(* IEC 61131-3 sources: Conveyor/test/Conveyor, 12 files *)

(* ---- ConveyorAutoStartupTest.st ---- *)
USING Simatic.Ax.Conveyor.Mocks;
USING Simatic.Ax.Conveyor;
USING AxUnit.Assert;
USING Simatic.Ax.AutomationBase;
USING MotorTests.Mocks;

NAMESPACE Simatic.Ax.Conveyor
    /// Tests for conveyor automatic startup behavior
    /// Verifies startup sequences, release conditions, and motor control during startup
    {TestFixture}
    CLASS ConveyorAutoStartupTest
        VAR
            conv : ConveyorBase;
            convStateless : ConveyorBase;
            mockMan : MockOperatingMode := (Mode := OperatingModes#Manual);
            mockManStateless : MockOperatingMode := (Mode := OperatingModes#Manual);
            relTrue : MockIsReleased_TRUE;
            relTrueStateless : MockIsReleased_TRUE;
            relFalse : MockIsReleased_FALSE;
            relFalseStateless : MockIsReleased_FALSE;
            autoStart : MockAutoStartup;
            autoStartStateless : MockAutoStartup;
            sensorMockQ_QRis_True : MockBinSignal := (QValue := TRUE, QRisValue := TRUE, QFalValue := FALSE);
            sensorMockQ_True : MockBinSignal := (QValue := TRUE, QRisValue := FALSE, QFalValue := FALSE);
            sensorMockQ_False : MockBinSignal := (QValue := FALSE, QRisValue := FALSE, QFalValue := FALSE);
            mockMotor : MockMotor;
            mockMotorStateless : MockMotor;
        END_VAR

        {TestSetup}
        METHOD PUBLIC Setup
            // Initialize stateless instances for each test
            conv := convStateless;
            mockMan := mockManStateless;
            relTrue := relTrueStateless;
            relFalse := relFalseStateless;
            autoStart := autoStartStateless;
            mockMotor := mockMotorStateless;
            mockMotor.Reset();
        END_METHOD

        {Test}
        METHOD PUBLIC Conveyor_Is_Stopped_InAutomatic_Without_Release
            // Arrange - Setup conveyor in automatic mode without release
            mockMan.mode := OperatingModes#Automatic;
            conv.Mode := mockMan;
            conv.Motor := mockMotor;
            conv.ExternalRelease := relTrue;
            conv.ExternalAutoStartup := autoStart;
            conv.StopSensor := sensorMockQ_False;
            autoStart.startupStatus := StartUpStatus#NotReleased;  // Not released

            // Verify setup is valid
            Equal(expected := FALSE, actual := HasConfigErrorTest(conv));

            // Act - Run cyclic execution
            conv.RunCyclic();

            // Assert - Motor should not be running without release
            Equal(expected := FALSE, actual := mockMotor.IsRunning());
        END_METHOD
        {Test}
        METHOD PUBLIC Conveyor_Is_Stopped_WhileStartingUp
            // Arrange - Setup conveyor during startup phase
            mockMan.mode := OperatingModes#Automatic;
            conv.Mode := mockMan;
            conv.Motor := mockMotor;
            conv.ExternalRelease := relTrue;
            autoStart.startupStatus := StartUpStatus#AutoStartingUp;  // Still starting up
            conv.StopSensor := sensorMockQ_False;
            conv.ExternalAutoStartup := autoStart;

            // Verify setup is valid
            Equal(expected := FALSE, actual := HasConfigErrorTest(conv));

            // Act - Run cyclic execution
            conv.RunCyclic();

            // Assert - Motor should not run during startup phase
            Equal(expected := FALSE, actual := mockMotor.IsRunning());
        END_METHOD
        {Test}
        METHOD PUBLIC Conveyor_Starts_After_AutoRelease
            // Arrange - Setup conveyor with auto-release completed
            mockMan.mode := OperatingModes#Automatic;
            conv.Mode := mockMan;
            conv.Motor := mockMotor;
            conv.ExternalRelease := relTrue;
            conv.StopSensor := sensorMockQ_False;
            autoStart.startupStatus := StartUpStatus#AutoStartedUp;  // Fully started up
            conv.ExternalAutoStartup := autoStart;

            // Mock timer to pass through immediately
            AxUnit.Mocking.Mock(NAME_OF(System.Timer.OffDelay), NAME_OF(Simatic.Ax.Mocks.OffDelayMock_pass_trough));

            // Act - Run cyclic execution
            conv.RunCyclic();

            // Assert - Motor should be running after auto-release
            Equal(expected := TRUE, actual := mockMotor.IsRunning());
        END_METHOD
        {Test}
        METHOD PUBLIC Conveyor_Stopps_after_loosing_release
            // Arrange - First start conveyor, then lose release
            THIS.Conveyor_Starts_After_AutoRelease();
            autoStart.startupStatus := StartUpStatus#NotReleased;  // Lose release

            // Verify setup is valid
            Equal(expected := FALSE, actual := HasConfigErrorTest(conv));

            // Act - Run cyclic execution after losing release
            conv.RunCyclic();

            // Assert - Motor should stop after losing release
            Equal(expected := FALSE, actual := mockMotor.IsRunning());
        END_METHOD
    END_CLASS

END_NAMESPACE

(* ---- ConveyorManualModeTest.st ---- *)
USING Simatic.Ax.Conveyor.Mocks;
USING Simatic.Ax.Conveyor;
USING AxUnit.Assert;
USING Simatic.Ax.AutomationBase;
USING MotorTests.Mocks;

NAMESPACE Simatic.Ax.Conveyor

    /// Tests for conveyor manual mode operation
    /// Verifies manual start/stop behavior, release conditions, and mode transitions
    {TestFixture}
    CLASS TestConveyorManualMode
        VAR
            conv : ConveyorBase;
            convStateless : ConveyorBase;
            mockMan : MockOperatingMode;
            mockManStateless : MockOperatingMode;
            relTrue : MockIsReleased_TRUE;
            relTrueStateless : MockIsReleased_TRUE;
            relFalse : MockIsReleased_FALSE;
            relFalseStateless : MockIsReleased_FALSE;
            StopSensor : MockBinSignal := (QValue := TRUE);
            mockMotor : MockMotor;
            mockMotorStateless : MockMotor;
        END_VAR

        {TestSetup}
        METHOD PUBLIC Setup
            // Initialize stateless instances for each test
            conv := convStateless;
            mockMan := mockManStateless;
            relTrue := relTrueStateless;
            relFalse := relFalseStateless;
            mockMotor := mockMotorStateless;
            mockMotor.Reset();
        END_METHOD

        {Test}
        METHOD PUBLIC ConveyorIsStoppedByDefault
            // Arrange - Setup conveyor in automatic mode with release
            conv.StopSensor := StopSensor;
            conv.Motor := mockMotor;
            mockMan.mode := OperatingModes#Automatic;
            conv.Mode := mockMan;
            conv.ExternalRelease := relTrue;

            // Verify configuration is valid
            Equal(expected := FALSE, actual := HasConfigErrorTest(conv));

            // Act - Run cyclic execution twice
            conv.RunCyclic();

            // Assert - Motor should remain stopped without explicit start command
            Equal(expected := FALSE, actual := mockMotor.IsRunning());

            // Act - Run cyclic again
            conv.RunCyclic();

            // Assert - Motor should still be stopped
            Equal(expected := FALSE, actual := mockMotor.IsRunning());
        END_METHOD
        {Test}
        METHOD PUBLIC Conveyor_InManualMode_RunReleasedOnManualStart
            // Arrange - Setup conveyor in manual mode with release
            conv.StopSensor := StopSensor;
            conv.Motor := mockMotor;
            conv.Mode := mockMan;  // Default mode is Manual
            conv.ExternalRelease := relTrue;

            // Act - Issue manual start command and run cyclic
            conv.StartManual();
            conv.RunCyclic();

            // Assert - Motor should be running after manual start
            Equal(expected := TRUE, actual := mockMotor.IsRunning());
        END_METHOD
        {Test}
        METHOD PUBLIC NotReleased_Conveyor_DoNotSetRunRelease
            // Arrange - Setup conveyor without release signal
            conv.StopSensor := StopSensor;
            conv.Motor := mockMotor;
            conv.Mode := mockMan;
            conv.ExternalRelease := relFalse;  // No release signal

            // Verify configuration is valid
            Equal(expected := FALSE, actual := HasConfigErrorTest(conv));

            // Act - Run cyclic, then issue manual start, then run cyclic again
            conv.RunCyclic();
            conv.StartManual();
            conv.RunCyclic();

            // Assert - Motor should not run without release signal
            Equal(expected := FALSE, actual := mockMotor.IsRunning());
        END_METHOD
        {Test}
        METHOD PUBLIC ConveyorManualRunning_Stops_when_release_signal_has_left
            // Arrange - Setup conveyor running in manual mode
            conv.StopSensor := StopSensor;
            conv.Motor := mockMotor;
            THIS.Conveyor_InManualMode_RunReleasedOnManualStart();

            // Act - Run cyclic while motor is running
            conv.RunCyclic();

            // Assert - Motor should still be running
            Equal(expected := TRUE, actual := mockMotor.IsRunning());

            // Act - Run cyclic again
            conv.RunCyclic();

            // Assert - Motor should still be running
            Equal(expected := TRUE, actual := mockMotor.IsRunning());

            // Act - Remove release signal and run cyclic
            conv.ExternalRelease := relFalse;
            conv.RunCyclic();

            // Assert - Motor should stop when release signal is lost
            Equal(expected := FALSE, actual := mockMotor.IsRunning());
        END_METHOD
        {Test}
        METHOD PUBLIC Conveyor_InAutomaticMode_IsNotRunReleasedOnManualStart
            // Arrange - Setup conveyor in automatic mode with release
            conv.StopSensor := StopSensor;
            conv.Motor := mockMotor;
            mockMan.mode := OperatingModes#Automatic;
            conv.Mode := mockMan;
            conv.ExternalRelease := relTrue;

            // Verify configuration is valid
            Equal(expected := FALSE, actual := HasConfigErrorTest(conv));

            // Act - Issue manual start command (should be ignored in automatic mode)
            conv.StartManual();
            conv.RunCyclic();

            // Assert - Motor should not run because manual start is ignored in automatic mode
            Equal(expected := FALSE, actual := mockMotor.IsRunning());
        END_METHOD
        {Test}
        METHOD PUBLIC ConveyorRunningInManualMode_Stops_on_Stop_Command
            // Arrange - Setup conveyor running in manual mode
            conv.StopSensor := StopSensor;
            conv.Motor := mockMotor;
            THIS.Conveyor_InManualMode_RunReleasedOnManualStart();

            // Act - Issue stop command and run cyclic
            conv.Stop();
            conv.RunCyclic();

            // Assert - Motor should stop after stop command
            Equal(expected := FALSE, actual := mockMotor.IsRunning());
        END_METHOD
    END_CLASS

END_NAMESPACE

(* ---- ConveyorMotorIntegrationTest.st ---- *)
USING AxUnit.Assert;
USING Simatic.Ax.Conveyor;
USING MotorTests.Mocks;

NAMESPACE ConveyorTests
    /// Integration tests for Conveyor with Motor
    {TestFixture}
    CLASS ConveyorMotorIntegrationTest
        VAR PROTECTED
            conveyor : ConveyorBase;
            conveyorStateless : ConveyorBase;
            motor : MockMotor;
            motorStateless : MockMotor;
        END_VAR

        {TestSetup}
        METHOD PUBLIC TestSetup
            conveyor := conveyorStateless;
            motor := motorStateless;
            motor.Reset();
        END_METHOD

        {Test}
        METHOD PUBLIC Test_ConveyorWithoutMotor_NoError
            // Arrange - No motor assigned

            // Act
            conveyor.RunCyclic();  // Init is now called automatically by RunCyclic

            // Assert - No motor calls when motor is NULL
            Equal(expected := 0, actual := motor.StartMotorCallCount);
        END_METHOD

        {Test}
        METHOD PUBLIC Test_ConveyorWithMotor_MotorInjected
            // Arrange
            conveyor.Motor := motor;

            // Act
            conveyor.RunCyclic();  // Init is now called automatically by RunCyclic

            // Assert - Motor is properly injected
            Equal(expected := TRUE, actual := (conveyor.Motor <> NULL));
        END_METHOD

        {Test}
        METHOD PUBLIC Test_MotorConfiguration_IsAccessible
            // Arrange & Act
            conveyor.Motor := motor;
            conveyor.AutomaticSpeed := 75.0;
            conveyor.Acceleration := 10.0;

            // Assert - Configuration is properly set
            Equal(expected := 75.0, actual := conveyor.AutomaticSpeed);
            Equal(expected := 10.0, actual := conveyor.Acceleration);
        END_METHOD

        {Test}
        METHOD PUBLIC Test_MotorConfiguration_SlowSpeed
            // Arrange
            conveyor.Motor := motor;
            conveyor.AutomaticSpeed := 75.0;
            conveyor.ManualSpeed := 30.0;

            // Act & Assert - Configuration is accessible
            Equal(expected := 75.0, actual := conveyor.AutomaticSpeed);
            Equal(expected := 30.0, actual := conveyor.ManualSpeed);
        END_METHOD

        {Test}
        METHOD PUBLIC Test_ConveyorStop_CallsStopMethod
            // Arrange
            conveyor.Motor := motor;
            Motor.StartMotor();

            // Act
            conveyor.Stop();

            // Assert - Stop method was called successfully
            Equal(expected := TRUE, actual := TRUE);  // Stop executed without error
        END_METHOD

        {Test}
        METHOD PUBLIC Test_IsMotorRunning_ReturnsMotorState
            // Arrange
            conveyor.Motor := motor;

            // Act & Assert - Motor not running
            Equal(expected := FALSE, actual := conveyor.ConveyorIsRunning());

            // Start motor
            Motor.StartMotor();

            // Act & Assert - Motor running
            Equal(expected := TRUE, actual := conveyor.ConveyorIsRunning());
        END_METHOD

        {Test}
        METHOD PUBLIC Test_MotorConfiguration_UsesCustomValues
            // Arrange
            conveyor.Motor := motor;
            conveyor.AutomaticSpeed := 80.0;
            conveyor.ManualSpeed := 25.0;
            conveyor.Acceleration := 15.0;
            conveyor.Deceleration := 20.0;

            // Act & Assert
            Equal(expected := 80.0, actual := conveyor.AutomaticSpeed);
            Equal(expected := 25.0, actual := conveyor.ManualSpeed);
            Equal(expected := 15.0, actual := conveyor.Acceleration);
            Equal(expected := 20.0, actual := conveyor.Deceleration);
        END_METHOD

        {Test}
        METHOD PUBLIC Test_MotorStopWithDeceleration
            // Arrange
            conveyor.Motor := motor;
            conveyor.Deceleration := 20.0;
            motor.FixedDeceleration := 20.0;
            Motor.StartMotor();

            // Act
            Motor.StopMotor();

            // Assert - Motor uses configured deceleration and stops
            Equal(expected := 20.0, actual := motor.FixedDeceleration);
            Equal(expected := FALSE, actual := motor.IsRunning());
        END_METHOD

        {Test}
        METHOD PUBLIC Test_IsMotorRunning_WithoutMotor_ReturnsFalse
            // Arrange
            conveyor.Motor := NULL;

            // Act & Assert
            Equal(expected := FALSE, actual := conveyor.ConveyorIsRunning());
        END_METHOD
    END_CLASS

    /// Tests for motor control logic
    {TestFixture}
    CLASS ConveyorMotorControlTest
        VAR PROTECTED
            conveyor : ConveyorBase;
            conveyorStateless : ConveyorBase;
            motor : MockMotor;
            motorStateless : MockMotor;
        END_VAR

        {TestSetup}
        METHOD PUBLIC TestSetup
            conveyor := conveyorStateless;
            motor := motorStateless;
            motor.Reset();
            conveyor.Motor := motor;
        END_METHOD

        {Test}
        METHOD PUBLIC Test_MockMotor_CanStartAndStop
            // Arrange
            conveyor.AutomaticSpeed := 75.0;
            conveyor.Deceleration := 15.0;

            // Act - Start motor
            Motor.StartMotor();

            // Assert - Motor started
            Equal(expected := TRUE, actual := motor.IsRunning());
            Equal(expected := 1, actual := motor.StartMotorCallCount);

            // Act - Stop motor
            Motor.StopMotor();

            // Assert - Motor stopped
            Equal(expected := FALSE, actual := motor.IsRunning());
            Equal(expected := 1, actual := motor.StopMotorCallCount);
        END_METHOD

        {Test}
        METHOD PUBLIC Test_MockMotor_TracksCallCounts
            // Arrange
            motor.TargetSpeed := 80.0;
            motor.FixedAcceleration := 12.0;
            motor.FixedDeceleration := 18.0;

            // Act
            Motor.StartMotor();
            Motor.StopMotor();

            // Assert - Call counts are tracked and properties are set
            Equal(expected := 1, actual := motor.StartMotorCallCount);
            Equal(expected := 1, actual := motor.StopMotorCallCount);
            Equal(expected := 80.0, actual := motor.TargetSpeed);
            Equal(expected := 12.0, actual := motor.FixedAcceleration);
            Equal(expected := 18.0, actual := motor.FixedDeceleration);
        END_METHOD

        {Test}
        METHOD PUBLIC Test_MockMotor_ResetClearsState
            // Arrange
            Motor.StartMotor();

            // Act
            motor.Reset();

            // Assert - All state cleared
            Equal(expected := FALSE, actual := motor.IsRunning());
            Equal(expected := 0, actual := motor.StartMotorCallCount);
            Equal(expected := 0, actual := motor.StopMotorCallCount);
            Equal(expected := 0.0, actual := motor.GetCurrentSpeed());
        END_METHOD
    END_CLASS
END_NAMESPACE

(* ---- ConveyorOccupiedStatus.st ---- *)
USING Simatic.Ax.Conveyor.Mocks;
USING Simatic.Ax.Conveyor;
USING AxUnit.Assert;
USING Simatic.Ax.AutomationBase;
USING MotorTests.Mocks;

NAMESPACE Simatic.Ax.Conveyor

    /// Tests for conveyor occupied status detection
    /// Verifies occupied state based on sensor coverage, operating mode, and startup status
    {TestFixture}
    CLASS ConveyorOccupiedStatus
        VAR
            conv : ConveyorBase;
            convStateless : ConveyorBase;
            mockOperatingMode : MockOperatingMode;
            mockOperatingModeStateless : MockOperatingMode;
            relTrue : MockIsReleased_TRUE;
            relTrueStateless : MockIsReleased_TRUE;
            relFalse : MockIsReleased_FALSE;
            relFalseStateless : MockIsReleased_FALSE;
            autoStart : MockAutoStartup;
            autoStartStateless : MockAutoStartup;
            sensorMockQ_QRis_True : MockBinSignal := (QValue := TRUE, QRisValue := TRUE, QFalValue := FALSE);
            sensorMockQ_True : MockBinSignal := (QValue := TRUE, QRisValue := FALSE, QFalValue := FALSE);
            sensorMockQ_False : MockBinSignal := (QValue := FALSE, QRisValue := FALSE, QFalValue := FALSE);
            convNext : MockingConveyor;
            convNextStateless : MockingConveyor;
            mockMotor : MockMotor;
            mockMotorStateless : MockMotor;
        END_VAR

        {TestSetup}
        METHOD PUBLIC Setup
            // Initialize stateless instances for each test
            conv := convStateless;
            mockOperatingMode := mockOperatingModeStateless;
            relTrue := relTrueStateless;
            relFalse := relFalseStateless;
            autoStart := autoStartStateless;
            convNext := convNextStateless;
            mockMotor := mockMotorStateless;
            mockMotor.Reset();
        END_METHOD

        METHOD PUBLIC SetupAutoStarted
            conv.StopSensor := sensorMockQ_False;
            conv.Motor := mockMotor;
            mockOperatingMode.mode := OperatingModes#Automatic;
            conv.Mode := mockOperatingMode;
            conv.Motor := mockMotor;
            conv.ExternalRelease := relTrue;
            conv.ExternalAutoStartup := autoStart;
            conv.NextConveyor := convNext;
            autoStart.startupStatus := StartUpStatus#AutoStartedUp;
        END_METHOD
        {Test}
        METHOD PUBLIC Conveyor_is_not_occupied_by_default
            // Arrange - Setup conveyor in auto-started state with no sensor coverage
            THIS.SetupAutoStarted();

            // Verify configuration is valid
            Equal(expected := FALSE, actual := HasConfigErrorTest(conv));

            // Act - Run cyclic execution
            conv.RunCyclic();

            // Assert - Conveyor should not be occupied without sensor coverage
            Equal(expected := FALSE, actual := conv.IsOccupied());
        END_METHOD
        {Test}
        METHOD PUBLIC Conveyor_Is_occupied_when_sensor_covered_and_automatic_is_on_while_next_is_not_rtr
            // Arrange - Setup conveyor in automatic mode with sensor covered
            THIS.SetupAutoStarted();
            conv.StopSensor := sensorMockQ_True;  // Sensor covered
            conv.Motor := mockMotor;
            // Next conveyor not ready to receive (default state)

            // Verify configuration is valid
            Equal(expected := FALSE, actual := HasConfigErrorTest(conv));

            // Act - Run cyclic execution
            conv.RunCyclic();

            // Assert - Conveyor should be occupied when sensor is covered in automatic mode
            Equal(expected := TRUE, actual := conv.IsOccupied());
        END_METHOD
        {Test}
        METHOD PUBLIC Conveyor_Ignores_occupied_state_when_in_manual
            // Arrange - Setup conveyor in manual mode with sensor covered
            THIS.SetupAutoStarted();
            conv.ExternalAutoStartup := NULL;
            conv.StopSensor := sensorMockQ_True;  // Sensor covered
            conv.Motor := mockMotor;
            mockOperatingMode.mode := OperatingModes#Manual;  // Manual mode

            // Verify configuration is valid
            Equal(expected := FALSE, actual := HasConfigErrorTest(conv));

            // Act - Run cyclic execution
            conv.RunCyclic();

            // Assert - Conveyor should not report occupied in manual mode (occupied detection disabled)
            Equal(expected := FALSE, actual := conv.IsOccupied());

        END_METHOD

        {Test}
        METHOD PUBLIC Conveyor_Is_occupied_when_sensor_covered_and_switch_to_automatic_while_next_is_not_rtr
            // Arrange - Setup conveyor with sensor covered, starting in manual mode
            conv.StopSensor := sensorMockQ_True;  // Sensor covered
            conv.Motor := mockMotor;
            mockOperatingMode.mode := OperatingModes#Manual;
            conv.Mode := mockOperatingMode;
            conv.ExternalRelease := relTrue;
            conv.ExternalAutoStartup := autoStart;
            conv.NextConveyor := convNext;

            // Act - Test in NotReleased state (manual mode)
            autoStart.startupStatus := StartUpStatus#NotReleased;
            conv.RunCyclic();

            // Assert - Not occupied in manual/not released state
            Equal(expected := FALSE, actual := conv.IsOccupied());

            // Act - Test during startup sequence
            autoStart.startupStatus := StartUpStatus#AutoStartingUp;
            conv.RunCyclic();

            // Assert - Not occupied during startup
            Equal(expected := FALSE, actual := conv.IsOccupied());

            // Act - Complete startup to automatic mode
            autoStart.startupStatus := StartUpStatus#AutoStartedUp;
            conv.RunCyclic();

            // Assert - Now occupied after fully started in automatic mode
            Equal(expected := TRUE, actual := conv.IsOccupied());
        END_METHOD
    END_CLASS

END_NAMESPACE

(* ---- ConveyorResetTest.st ---- *)
USING Simatic.Ax.AutomationBase;
USING AxUnit.Assert;
USING Simatic.Ax.Conveyor;
USING Simatic.Ax.Conveyor.Mocks;
USING Simatic.Ax.AutomationBase;
USING MotorTests.Mocks;

NAMESPACE Simatic.Ax.Conveyor.Tests

    {TestFixture}
    CLASS ConveyorResetTest
        VAR
            conveyor : ConveyorBase;
            conveyorStateless : ConveyorBase;
            mockMotor : MockMotor;
            mockMotorStateless : MockMotor;
            mockMode : MockOperatingMode := (Mode := OperatingModes#Manual);
            mockModeStateless : MockOperatingMode := (Mode := OperatingModes#Manual);
            mockRelease : MockIsReleased_TRUE;
            mockReleaseStateless : MockIsReleased_TRUE;
            mockAutoStartup : MockAutoStartup;
            mockAutoStartupStateless : MockAutoStartup;
            mockResetManager : MockResetManager;
            mockResetManagerStateless : MockResetManager;
            sensorMockQ_True : MockBinSignal := (QValue := TRUE, QRisValue := FALSE, QFalValue := FALSE);
            sensorMockQ_False : MockBinSignal := (QValue := FALSE, QRisValue := FALSE, QFalValue := FALSE);
        END_VAR

        {TestSetup}
        METHOD PUBLIC Setup
            // Reset to stateless instances for test isolation
            conveyor := conveyorStateless;
            mockMotor := mockMotorStateless;
            mockMotor.Reset();
            mockMode := mockModeStateless;
            mockRelease := mockReleaseStateless;
            mockAutoStartup := mockAutoStartupStateless;
            mockResetManager := mockResetManagerStateless;
            mockResetManager.Reset();

            // Configure conveyor
            conveyor.StopSensor := sensorMockQ_False;
            conveyor.Motor := mockMotor;
            conveyor.ExternalRelease := mockRelease;
            conveyor.Mode := mockMode;
            conveyor.ExternalAutoStartup := mockAutoStartup;
            conveyor.ResetCommand := mockResetManager;

            // Set default states
            mockMode.mode := OperatingModes#Automatic;
            mockAutoStartup.startupStatus := StartUpStatus#AutoStartedUp;

            // Initialize conveyor by calling RunCyclic (triggers InitUser)
            conveyor.RunCyclic();
        END_METHOD

        {Test}
        METHOD PUBLIC Test_ResetFault_ClearsManualStartFlag
            // Arrange
            mockMode.mode := OperatingModes#Manual;
            mockAutoStartup.startupStatus := StartUpStatus#Manual;
            conveyor.RunCyclic();
            conveyor.StartManual();
            conveyor.RunCyclic();
            Equal(expected := TRUE, actual := Conveyor.ConveyorIsRunning());
            conveyor.SetError(errorState := WORD#16#8199, errorText := 'any error');

            // Verify motor is running
            Equal(expected := TRUE, actual := mockMotor.StartMotorCallCount > 0);

            // Act - trigger reset via ResetManager
            mockResetManager.ResetCommandActive := TRUE;
            conveyor.RunCyclic();

            // Assert - manual start flag should be cleared
            mockResetManager.ResetCommandActive := FALSE;
            conveyor.RunCyclic();
            Equal(expected := TRUE, actual := mockMotor.StopMotorCallCount > 0);
        END_METHOD

        {Test}
        METHOD PUBLIC Test_ResetFault_AllowsAutoRestart
            // Arrange - setup conveyor with material
            conveyor.StopSensor := sensorMockQ_True;
            conveyor.RunCyclic();

            // Simulate error
            conveyor.SetError(errorState := WORD#16#8001, errorText := 'Test error');

            // Act - trigger reset via ResetManager
            mockResetManager.ResetCommandActive := TRUE;
            conveyor.RunCyclic();

            // Assert - conveyor should be able to auto-restart after reset
            // The auto-release flags are NOT cleared, allowing automatic restart
            mockResetManager.ResetCommandActive := FALSE;
            conveyor.RunCyclic();
            conveyor.TriggerStartInAutomatic();
            conveyor.RunCyclic();
            Equal(expected := TRUE, actual := mockMotor.StartMotorCallCount > 0);
        END_METHOD

        {Test}
        METHOD PUBLIC Test_ResetFault_AllowsNormalOperationAfterReset
            // Arrange - trigger reset
            mockResetManager.ResetCommandActive := TRUE;
            conveyor.RunCyclic();
            mockResetManager.ResetCommandActive := FALSE;

            // Act - simulate normal operation
            conveyor.StopSensor := sensorMockQ_True;
            conveyor.RunCyclic();
            conveyor.TriggerStartInAutomatic();
            conveyor.RunCyclic();

            // Assert - conveyor should be able to start normally
            Equal(expected := TRUE, actual := mockMotor.StartMotorCallCount > 0);
        END_METHOD

        {Test}
        METHOD PUBLIC Test_ResetFault_CanBeCalledMultipleTimes
            // Act - trigger reset multiple times via ResetManager
            mockResetManager.ResetCommandActive := TRUE;
            conveyor.RunCyclic();
            conveyor.RunCyclic();
            conveyor.RunCyclic();

            // Assert - should not cause any issues
            mockResetManager.ResetCommandActive := FALSE;
            conveyor.RunCyclic();
            Equal(expected := FALSE, actual := conveyor.HasError());
        END_METHOD
        {Test}
        METHOD PUBLIC Test_ResetFault_WithNullMotor_DoesNotCrash
            // Arrange
            conveyor.Motor := NULL;

            // Act & Assert - should not crash when reset is triggered
            mockResetManager.ResetCommandActive := TRUE;
            conveyor.RunCyclic();
            mockResetManager.ResetCommandActive := FALSE;
            conveyor.RunCyclic();
            Equal(expected := FALSE, actual := conveyor.HasError());
        END_METHOD

        {Test}
        METHOD PUBLIC Test_ResetFault_ClearsErrorState
            // Arrange - simulate an error condition
            conveyor.SetError(errorState := WORD#16#8001, errorText := 'Test error');
            Equal(expected := TRUE, actual := conveyor.HasError());

            // Act - trigger reset via ResetManager
            mockResetManager.ResetCommandActive := TRUE;
            conveyor.RunCyclic();

            // Assert - error should be cleared
            Equal(expected := FALSE, actual := conveyor.HasError());
        END_METHOD

        // {Test}
        // METHOD PUBLIC Test_ResetFault_BlockedWhenSensorStillCovered
        //     // Arrange - simulate sensor blocked during delivering
        //     sensorMockQ_True.QValue := TRUE;
        //     conveyor.StopSensor := sensorMockQ_True;
        //     conveyor.RunCyclic();
        //     conveyor.TriggerStartInAutomatic();
        //     conveyor.RunCyclic();

        //     // Simulate error condition
        //     conveyor.SetError(errorState := WORD#16#8001, errorText := 'Sensor blocked');
        //     Equal(expected := TRUE, actual := conveyor.HasError());

        //     // Act - try to reset while sensor is still covered via ResetManager
        //     mockResetManager.ResetCommandActive := TRUE;
        //     conveyor.RunCyclic();

        //     // Assert - error should NOT be cleared because sensor is still blocked
        //     Equal(expected := TRUE, actual := conveyor.HasError());
        // END_METHOD

        {Test}
        METHOD PUBLIC Test_ResetFault_AllowedWhenSensorCleared
            // Arrange - simulate sensor blocked, then cleared
            sensorMockQ_True.QValue := TRUE;
            conveyor.StopSensor := sensorMockQ_True;
            conveyor.RunCyclic();
            conveyor.TriggerStartInAutomatic();
            conveyor.RunCyclic();

            // Simulate error condition
            conveyor.SetError(errorState := WORD#16#8001, errorText := 'Sensor blocked');
            Equal(expected := TRUE, actual := conveyor.HasError());

            // Clear the sensor
            conveyor.StopSensor := sensorMockQ_False;
            conveyor.RunCyclic();

            // Act - reset after sensor is cleared via ResetManager
            mockResetManager.ResetCommandActive := TRUE;
            conveyor.RunCyclic();

            // Assert - error should be cleared now
            Equal(expected := FALSE, actual := conveyor.HasError());
        END_METHOD
    END_CLASS

END_NAMESPACE

(* ---- EndOfLineConveyorTest.st ---- *)
USING Simatic.Ax.Conveyor.Mocks;
USING Simatic.Ax.Conveyor;
USING AxUnit.Assert;
USING Simatic.Ax.AutomationBase;
USING MotorTests.Mocks;

NAMESPACE Simatic.Ax.Conveyor

    /// Tests for end-of-line conveyor behavior with NullReceiver
    /// Verifies that the last conveyor in a line can complete transfers without a next conveyor
    {TestFixture}
    CLASS EndOfLineConveyorTest
        VAR
            conv : ConveyorBase;
            convStateless : ConveyorBase;
            sensor : MockBinSignal;
            sensorStateless : MockBinSignal;
            relTrue : MockIsReleased_TRUE;
            relTrueStateless : MockIsReleased_TRUE;
            autoStart : MockAutoStartup := (startupStatus := StartUpStatus#AutoStartedUp);
            autoStartStateless : MockAutoStartup := (startupStatus := StartUpStatus#AutoStartedUp);
            mode : MockOperatingMode;
            modeStateless : MockOperatingMode;
            mockMotor : MockMotor;
            mockMotorStateless : MockMotor;
            nullReceiver : NullReceiver;
            nullReceiverStateless : NullReceiver;
        END_VAR

        {TestSetup}
        METHOD PUBLIC TestSetup
            // Initialize stateless instances for each test
            conv := convStateless;
            sensor := sensorStateless;
            relTrue := relTrueStateless;
            autoStart := autoStartStateless;
            mode := modeStateless;
            mockMotor := mockMotorStateless;
            mockMotor.Reset();
            nullReceiver := nullReceiverStateless;

            // Setup end-of-line conveyor (no NextConveyor configured)
            conv.NextConveyor := NULL;  // End of line - will use NullReceiver
            conv.StopSensor := sensor;
            conv.Motor := mockMotor;
            conv.ExternalRelease := relTrue;
            conv.ExternalAutoStartup := autoStart;
            conv.Mode := mode;
            mode.mode := OperatingModes#Automatic;
            conv.OffDelayTime := T#2s;
            AxUnit.Mocking.Mock('System.Timer.OffDelay', 'Simatic.Ax.Mocks.OffDelayMock_pass_trough');
        END_METHOD

        {Test}
        METHOD PUBLIC EndOfLine_conveyor_starts_transfer_when_sensor_covered
            // Arrange - End of line conveyor with no next conveyor
            sensor.QValue := FALSE;

            // Act - Run cyclic to initialize
            conv.RunCyclic();

            // Act - Item arrives on sensor
            sensor.QValue := TRUE;
            conv.RunCyclic();

            // Assert - Conveyor should start transfer even without next conveyor
            Equal(expected := TRUE, actual := conv.IsOccupied());
            Equal(expected := TRUE, actual := conv.DeliverStatus() = DeliverState#Delivering);
            Equal(expected := TRUE, actual := mockMotor.IsRunning());
        END_METHOD

        {Test}
        METHOD PUBLIC EndOfLine_conveyor_continues_running_until_item_leaves
            // Arrange - Start with item on sensor
            THIS.EndOfLine_conveyor_starts_transfer_when_sensor_covered();

            // Assert - Motor should be running
            Equal(expected := TRUE, actual := mockMotor.IsRunning());

            // Act - Continue running while item is on sensor
            conv.RunCyclic();
            Equal(expected := TRUE, actual := mockMotor.IsRunning());

            conv.RunCyclic();
            Equal(expected := TRUE, actual := mockMotor.IsRunning());

            // Act - Item leaves sensor (transfer complete)
            sensor.QValue := FALSE;
            conv.RunCyclic();

            // Assert - Transfer should be complete, motor still running due to off-delay
            Equal(expected := TRUE, actual := conv.DeliverStatus() = DeliverState#Idle);
            Equal(expected := FALSE, actual := conv.IsOccupied());
            Equal(expected := TRUE, actual := mockMotor.IsRunning());
        END_METHOD

        {Test}
        METHOD PUBLIC EndOfLine_conveyor_stops_after_offdelay_expires
            // Arrange - Complete transfer and wait for off-delay
            THIS.EndOfLine_conveyor_continues_running_until_item_leaves();

            // Assert - Motor still running after transfer
            Equal(expected := TRUE, actual := mockMotor.IsRunning());

            // Act - Simulate off-delay timer expiring
            AxUnit.Mocking.Mock('System.Timer.OffDelay', 'Simatic.Ax.Mocks.OffDelayMock_false');
            conv.RunCyclic();

            // Assert - Motor should stop after off-delay expires
            Equal(expected := FALSE, actual := mockMotor.IsRunning());
        END_METHOD
{Test}
METHOD PUBLIC NullReceiver_always_signals_ReadyToReceive
    // Arrange - NullReceiver already initialized in TestSetup

            // Act & Assert - NullReceiver should always return ReadyToReceive
            Equal(expected := TRUE, actual := nullReceiver.ReceiveStatus() = ReceiveState#ReadyToReceive);

            // Call multiple times to ensure consistent behavior
            Equal(expected := TRUE, actual := nullReceiver.ReceiveStatus() = ReceiveState#ReadyToReceive);
            Equal(expected := TRUE, actual := nullReceiver.ReceiveStatus() = ReceiveState#ReadyToReceive);
        END_METHOD
    END_CLASS

END_NAMESPACE

(* ---- ExtendRunningForConveyorTest.st ---- *)
USING Simatic.Ax.Conveyor.Mocks;
USING Simatic.Ax.Conveyor;
USING AxUnit.Assert;
USING Simatic.Ax.AutomationBase;
USING MotorTests.Mocks;

NAMESPACE Simatic.Ax.Conveyor

    /// Tests for extended running behavior of conveyor
    /// Verifies motor continues running after base position until timeout
    {TestFixture}
    CLASS ExtendRunningForConveyorTest
        VAR
            conv : ConveyorBase;
            convStateless : ConveyorBase;
            nextConv : MockingConveyor;
            nextConvStateless : MockingConveyor;
            sensor : MockBinSignal;
            sensorStateless : MockBinSignal;
            relTrue : MockIsReleased_TRUE;
            relTrueStateless : MockIsReleased_TRUE;
            relFalse : MockIsReleased_FALSE;
            relFalseStateless : MockIsReleased_FALSE;
            autoStart : MockAutoStartup := (startupStatus := StartUpStatus#AutoStartedUp);
            autoStartStateless : MockAutoStartup := (startupStatus := StartUpStatus#AutoStartedUp);
            mode : MockOperatingMode;
            modeStateless : MockOperatingMode;
            mockMotor : MockMotor;
            mockMotorStateless : MockMotor;
        END_VAR

        {TestSetup}
        METHOD PUBLIC TestSetup
            // Initialize stateless instances for each test
            conv := convStateless;
            nextConv := nextConvStateless;
            sensor := sensorStateless;
            relTrue := relTrueStateless;
            relFalse := relFalseStateless;
            autoStart := autoStartStateless;
            mode := modeStateless;
            mockMotor := mockMotorStateless;
            mockMotor.Reset();

            // Setup conveyor configuration
            conv.NextConveyor := nextConv;
            conv.StopSensor := sensor;
            conv.Motor := mockMotor;
            conv.ExternalRelease := relTrue;
            conv.Mode := mode;
        END_METHOD
        {Test}
        METHOD PUBLIC Conveyor_Stopps_after_base_position_run_after_timeout
            // Arrange - Setup conveyor in manual mode, not released
            conv.ExternalAutoStartup := autoStart;
            autoStart.startupStatus := StartUpStatus#NotReleased;

            // Mock timer to pass through immediately (no delay)
            AxUnit.Mocking.Mock('System.Timer.OffDelay', 'Simatic.Ax.Mocks.OffDelayMock_pass_trough');

            mode.mode := OperatingModes#Manual;
            sensor.QValue := FALSE;  // No item on sensor

            // Act - Run cyclic in manual mode
            conv.RunCyclic();

            // Assert - Motor should not be running in manual mode without release
            Equal(expected := FALSE, actual := mockMotor.IsRunning());

            // Act - Switch to automatic mode and complete startup
            mode.mode := OperatingModes#Automatic;
            autoStart.startupStatus := StartUpStatus#AutoStartedUp;
            conv.RunCyclic();

            // Assert - Motor should start running after switching to automatic with completed startup
            Equal(expected := TRUE, actual := mockMotor.IsRunning());
        END_METHOD
    END_CLASS

END_NAMESPACE

(* ---- MotorRunsDuringDeliveringTest.st ---- *)
USING Simatic.Ax.Conveyor.Mocks;
USING Simatic.Ax.Conveyor;
USING AxUnit.Assert;
USING Simatic.Ax.AutomationBase;
USING MotorTests.Mocks;

NAMESPACE Simatic.Ax.Conveyor

    /// Tests for motor behavior during Delivering state
    /// Verifies that motor continues running during transfer regardless of next conveyor state changes
    {TestFixture}
    CLASS MotorRunsDuringDeliveringTest
        VAR
            conv : ConveyorBase;
            convStateless : ConveyorBase;
            nextConv : MockingConveyor;
            nextConvStateless : MockingConveyor;
            sensor : MockBinSignal;
            sensorStateless : MockBinSignal;
            relTrue : MockIsReleased_TRUE;
            relTrueStateless : MockIsReleased_TRUE;
            autoStart : MockAutoStartup := (startupStatus := StartUpStatus#AutoStartedUp);
            autoStartStateless : MockAutoStartup := (startupStatus := StartUpStatus#AutoStartedUp);
            mode : MockOperatingMode;
            modeStateless : MockOperatingMode;
            mockMotor : MockMotor;
            mockMotorStateless : MockMotor;
        END_VAR

        {TestSetup}
        METHOD PUBLIC TestSetup
            // Initialize stateless instances for each test
            conv := convStateless;
            nextConv := nextConvStateless;
            sensor := sensorStateless;
            relTrue := relTrueStateless;
            autoStart := autoStartStateless;
            mode := modeStateless;
            mockMotor := mockMotorStateless;
            mockMotor.Reset();

            // Setup conveyor configuration
            conv.NextConveyor := nextConv;
            conv.StopSensor := sensor;
            conv.Motor := mockMotor;
            conv.ExternalRelease := relTrue;
            conv.ExternalAutoStartup := autoStart;
            conv.Mode := mode;
            mode.mode := OperatingModes#Automatic;
            conv.OffDelayTime := T#2s;
            AxUnit.Mocking.Mock('System.Timer.OffDelay', 'Simatic.Ax.Mocks.OffDelayMock_pass_trough');
        END_METHOD

        {Test}
        METHOD PUBLIC Motor_continues_running_during_Delivering_when_next_conveyor_changes_state
            // Arrange - Setup conveyor with sensor covered and next conveyor ready
            nextConv.RTR := ReceiveState#ReadyToReceive;
            sensor.QValue := TRUE;  // Item on sensor

            // Act - Run cyclic execution to start transfer
            conv.RunCyclic();

            // Assert - Motor should be running and transfer in progress
            Equal(expected := TRUE, actual := mockMotor.IsRunning());
            Equal(expected := TRUE, actual := conv.DeliverStatus() = DeliverState#Delivering);

            // Act - Next conveyor changes state to Receiving (simulating material arriving)
            nextConv.RTR := ReceiveState#Receiving;
            conv.RunCyclic();

            // Assert - Motor should STILL be running despite next conveyor state change
            Equal(expected := TRUE, actual := mockMotor.IsRunning());
            Equal(expected := TRUE, actual := conv.DeliverStatus() = DeliverState#Delivering);

            // Act - Continue running while sensor still covered (transfer ongoing)
            conv.RunCyclic();

            // Assert - Motor should continue running during transfer
            Equal(expected := TRUE, actual := mockMotor.IsRunning());
            Equal(expected := TRUE, actual := conv.DeliverStatus() = DeliverState#Delivering);
        END_METHOD

        {Test}
        METHOD PUBLIC Motor_continues_running_during_Delivering_over_multiple_cycles
            // Arrange - Setup conveyor with sensor covered and next conveyor ready
            nextConv.RTR := ReceiveState#ReadyToReceive;
            sensor.QValue := TRUE;  // Item on sensor

            // Act - Run cyclic execution to start transfer
            conv.RunCyclic();

            // Assert - Transfer should be in progress
            Equal(expected := TRUE, actual := conv.DeliverStatus() = DeliverState#Delivering);
            Equal(expected := TRUE, actual := mockMotor.IsRunning());

            // Act - Run multiple cycles while in Delivering
            conv.RunCyclic();
            Equal(expected := TRUE, actual := mockMotor.IsRunning());

            conv.RunCyclic();
            Equal(expected := TRUE, actual := mockMotor.IsRunning());

            conv.RunCyclic();
            Equal(expected := TRUE, actual := mockMotor.IsRunning());

            conv.RunCyclic();
            Equal(expected := TRUE, actual := mockMotor.IsRunning());

            // Assert - Motor should remain running throughout the transfer
            Equal(expected := TRUE, actual := conv.DeliverStatus() = DeliverState#Delivering);
        END_METHOD

        {Test}
        METHOD PUBLIC Motor_stops_only_after_transfer_completes_and_offdelay_expires
            // Arrange - Setup conveyor with sensor covered and next conveyor ready
            nextConv.RTR := ReceiveState#ReadyToReceive;
            sensor.QValue := TRUE;  // Item on sensor

            // Act - Run cyclic execution to start transfer
            conv.RunCyclic();
            Equal(expected := TRUE, actual := mockMotor.IsRunning());

            // Act - Item leaves sensor (transfer completes)
            sensor.QValue := FALSE;
            conv.RunCyclic();

            // Assert - Transfer should be complete, motor still running due to off-delay
            Equal(expected := TRUE, actual := conv.DeliverStatus() = DeliverState#Idle);
            Equal(expected := TRUE, actual := mockMotor.IsRunning());

            // Act - Simulate off-delay timer expiring
            AxUnit.Mocking.Mock('System.Timer.OffDelay', 'Simatic.Ax.Mocks.OffDelayMock_false');
            nextConv.RTR := ReceiveState#Idle;
            conv.RunCyclic();

            // Assert - Now motor should stop after off-delay expires
            Equal(expected := FALSE, actual := mockMotor.IsRunning());
        END_METHOD
    END_CLASS

END_NAMESPACE

(* ---- ReceiveFromPreviousConveyor.st ---- *)
USING Simatic.Ax.Conveyor.Mocks;
USING Simatic.Ax.Conveyor;
USING AxUnit.Assert;
USING Simatic.Ax.AutomationBase;
USING MotorTests.Mocks;

NAMESPACE Simatic.Ax.Conveyor

    /// Tests for receiving items from previous conveyor
    /// Verifies conveyor starts when previous conveyor signals ready to deliver or transfer in progress
    {TestFixture}
    CLASS ReceiveFromPreviousConveyor
        VAR
            conv, convStateless : ConveyorBase;
            nextConv, nextConvStateless : MockingConveyor;
            prevConv, prevConvStateless : MockingConveyor;
            sensor, sensorStateless : MockBinSignal;
            relTrue,  relTrueStateless : MockIsReleased_TRUE;
            relFalse, relFalseStateless : MockIsReleased_FALSE;
            autoStart, autoStartStateless : MockAutoStartup := (startupStatus := StartUpStatus#AutoStartedUp);
            mode, modeStateless : MockOperatingMode;
            mockMotor, mockMotorStateless : MockMotor;
        END_VAR

        {TestSetup}
        METHOD PUBLIC TestSetup
            // Initialize stateless instances for each test
            conv := convStateless;
            nextConv := nextConvStateless;
            prevConv := prevConvStateless;
            sensor := sensorStateless;
            relTrue := relTrueStateless;
            relFalse := relFalseStateless;
            autoStart := autoStartStateless;
            mode := modeStateless;
            mockMotor := mockMotorStateless;
            mockMotor.Reset();

            conv.NextConveyor := nextConv;
            conv.PrevConveyor := prevConv;
            conv.StopSensor := sensor;
            conv.Motor := mockMotor;
            conv.ExternalRelease := relTrue;
            conv.ExternalAutoStartup := autoStart;
            conv.StopSensor := sensor;
            conv.Motor := mockMotor;
            conv.Mode := mode;
            conv.Motor := mockMotor;
            mode.mode := OperatingModes#Automatic;
            AxUnit.Mocking.Mock('System.Timer.OffDelay', 'Simatic.Ax.Mocks.OffDelayMock_pass_trough');

        END_METHOD

        {Test}
        METHOD PUBLIC Idle_Conveyor_Starts_direct_On_Previous_Conveyor_is_ReadyToDeilver
            VAR_TEMP
                motorIsReleased : BOOL;
            END_VAR

            // Arrange - Setup conveyor with no sensor coverage, fully started
            sensor.QValue := FALSE;
            autoStart.startupStatus := StartUpStatus#AutoStartedUp;

            // Act - Run cyclic for initial home position run
            conv.RunCyclic();

            // Assert - Motor should be running for home position
            Equal(expected := TRUE, actual := mockMotor.IsRunning());

            // Act - Simulate home position run finished (off delay expires)
            AxUnit.Mocking.Mock('System.Timer.OffDelay', 'Simatic.Ax.Mocks.OffDelayMock_false');
            conv.RunCyclic();
            motorIsReleased := mockMotor.IsRunning();

            // Assert - Motor should stop after home position run completes
            Equal(expected := FALSE, actual := motorIsReleased);

            // Act - Previous conveyor announces ready to deliver
            AxUnit.Mocking.Mock('System.Timer.OffDelay', 'Simatic.Ax.Mocks.OffDelayMock_pass_trough');
            prevConv.RTD := DeliverState#ReadyToDeliver;
            conv.RunCyclic();

            // Assert - Motor should start immediately when previous conveyor is ready to deliver
            Equal(expected := TRUE, actual := mockMotor.IsRunning());

        END_METHOD

        {Test}
        METHOD PUBLIC Idle_Conveyor_Starts_direct_On_Previous_Conveyor_is_Delivering
            VAR_TEMP
                motorIsReleased : BOOL;
            END_VAR

            // Arrange - Setup conveyor with no sensor coverage, fully started
            sensor.QValue := FALSE;
            autoStart.startupStatus := StartUpStatus#AutoStartedUp;

            // Act - Run cyclic for initial home position run
            conv.RunCyclic();

            // Assert - Motor should be running for home position
            Equal(expected := TRUE, actual := mockMotor.IsRunning());

            // Act - Simulate home position run finished (off delay expires)
            AxUnit.Mocking.Mock('System.Timer.OffDelay', 'Simatic.Ax.Mocks.OffDelayMock_false');
            conv.RunCyclic();
            motorIsReleased := mockMotor.IsRunning();

            // Assert - Motor should stop after home position run completes
            Equal(expected := FALSE, actual := motorIsReleased);

            // Act - Previous conveyor announces transfer in progress
            AxUnit.Mocking.Mock('System.Timer.OffDelay', 'Simatic.Ax.Mocks.OffDelayMock_pass_trough');
            prevConv.RTD := DeliverState#Delivering;
            conv.RunCyclic();

            // Assert - Motor should start immediately when previous conveyor has transfer in progress
            Equal(expected := TRUE, actual := mockMotor.IsRunning());

        END_METHOD
    END_CLASS

END_NAMESPACE

(* ---- StopPositionTest.st ---- *)
USING Simatic.Ax.Conveyor.Mocks;
USING Simatic.Ax.Conveyor;
USING AxUnit.Assert;
USING Simatic.Ax.AutomationBase;

NAMESPACE Simatic.Ax.Conveyor

    /// Tests for stop position occupied detection
    /// Verifies occupied state based on sensor and equipment startup status
    {TestFixture}
    CLASS StopPositionTest
        VAR
            stop : StopPosition;
            stopStateless : StopPosition;
            sens : MockBinSignal;
            sensStateless : MockBinSignal;
            conv : MockingConveyor;
            convStateless : MockingConveyor;
            eq : MockEquiment;
            eqStateless : MockEquiment;
        END_VAR

        {TestSetup}
        METHOD PUBLIC TestSetup
            // Initialize stateless instances for each test
            stop := stopStateless;
            sens := sensStateless;
            conv := convStateless;
            eq := eqStateless;
        END_METHOD

        METHOD PUBLIC Setup
            stop.Equipment := eq;
            stop.Deliverer := conv;
            stop.StopSensor := sens;
            ;
        END_METHOD

        {Test}
        METHOD PUBLIC StopPos_is_not_occupied_when_Q_Sensor_False
            // Arrange - Setup stop position with sensor not covered
            THIS.Setup();
            sens.QValue := FALSE;

            // Act - Evaluate stop position
            stop.EvaluateStopPos();

            // Assert - Stop position should not be occupied without sensor coverage
            Equal(expected := FALSE, actual := stop.IsOccupied());
        END_METHOD

        {Test}
        METHOD PUBLIC StopPos_is_not_occupied_when_Q_Sensor_False_And_Equipment_in_automatic
            // Arrange - Setup stop position with sensor not covered, equipment started
            THIS.Setup();
            sens.QValue := FALSE;
            eq.MockStatus := StartUpStatus#AutoStartedUp;

            // Act - Evaluate stop position
            stop.EvaluateStopPos();

            // Assert - Stop position should not be occupied without sensor coverage (even if started)
            Equal(expected := FALSE, actual := stop.IsOccupied());
        END_METHOD

        {Test}
        METHOD PUBLIC StopPos_is_not_occupied_when_Q_Sensor_True_and_starting_up
            // Arrange - Setup stop position with sensor covered but equipment starting up
            THIS.Setup();
            sens.QValue := TRUE;
            eq.MockStatus := StartUpStatus#AutoStartingUp;

            // Act - Evaluate stop position
            stop.EvaluateStopPos();

            // Assert - Stop position should not be occupied during startup (ignore sensor)
            Equal(expected := FALSE, actual := stop.IsOccupied());
        END_METHOD

        {Test}
        METHOD PUBLIC StopPos_is_not_occupied_when_Q_Sensor_True_and_not_released
            // Arrange - Setup stop position with sensor covered but equipment not released
            THIS.Setup();
            sens.QValue := TRUE;
            eq.MockStatus := StartUpStatus#NotReleased;

            // Act - Evaluate stop position
            stop.EvaluateStopPos();

            // Assert - Stop position should not be occupied without release (ignore sensor)
            Equal(expected := FALSE, actual := stop.IsOccupied());
        END_METHOD

        {Test}
        METHOD PUBLIC StopPos_is_occupied_when_Q_Sensor_True_and_is_released
            // Arrange - Setup stop position with sensor covered and equipment started
            THIS.Setup();
            sens.QValue := TRUE;
            eq.MockStatus := StartUpStatus#AutoStartedUp;

            // Act - Evaluate stop position
            stop.EvaluateStopPos();

            // Assert - Stop position should be occupied when sensor covered and equipment started
            Equal(expected := TRUE, actual := stop.IsOccupied());
        END_METHOD

        {Test}
        METHOD PUBLIC Uncover_Sensor_while_equipment_is_still_started_up_keeps_occupied
            // Arrange - Setup stop position that was occupied
            THIS.Setup();
            THIS.StopPos_is_occupied_when_Q_Sensor_True_and_is_released();

            // Act - Sensor becomes uncovered but equipment still started
            sens.QValue := FALSE;
            eq.MockStatus := StartUpStatus#AutoStartedUp;
            stop.EvaluateStopPos();

            // Assert - Stop position should remain occupied (latched state)
            Equal(expected := TRUE, actual := stop.IsOccupied());
        END_METHOD

        {Test}
        METHOD PUBLIC Stored_Occuoied_removes_when_state_Changes_from_StartingUp_to_StartedUp
            // Arrange - Setup stop position that was occupied
            THIS.Setup();
            THIS.StopPos_is_occupied_when_Q_Sensor_True_and_is_released();

            // Act - Sensor uncovered and equipment transitions to starting up
            sens.QValue := FALSE;
            eq.MockStatus := StartUpStatus#AutoStartingUp;

            // Assert - Stop position should still be occupied (latched)
            Equal(expected := TRUE, actual := stop.IsOccupied());

            // Act - Evaluate and then complete startup
            stop.EvaluateStopPos();
            eq.MockStatus := StartUpStatus#AutoStartedUp;

            // Assert - Occupied state should clear after startup cycle completes
            Equal(expected := FALSE, actual := stop.IsOccupied());
        END_METHOD
    END_CLASS

END_NAMESPACE

(* ---- TransportIntegrativeTest.st ---- *)
USING Simatic.Ax.Conveyor.Mocks;
USING Simatic.Ax.Conveyor;
USING AxUnit.Assert;
USING Simatic.Ax.AutomationBase;
NAMESPACE Simatic.Ax.Conveyor

    /// Integration tests for transport control logic
    /// Verifies interaction between ReadyToDeliver, ReadyToReceive, and StopPosition components
    {TestFixture}
    CLASS TransportIntegrativeTest
        VAR
            _rtd : ReadyToDeliver;
            _rtdStateless : ReadyToDeliver;
            _rtr : ReadyToReceive;
            _rtrStateless : ReadyToReceive;
            _stop : StopPosition;
            _stopStateless : StopPosition;
            conv : MockingConveyor;
            convStateless : MockingConveyor;
            eq : MockEquiment;
            eqStateless : MockEquiment;
            stopsensor : MockBinSignal;
            stopsensorStateless : MockBinSignal;
            nextConv : MockingConveyor;
            nextConvStateless : MockingConveyor;
            prevConv : MockingConveyor;
            prevConvStateless : MockingConveyor;
            _internalDeliverState : DeliverState;
            _internalReceiveState : ReceiveState;
        END_VAR

        {TestSetup}
        METHOD PUBLIC TestSetup
            // Initialize stateless instances for each test
            _rtd := _rtdStateless;
            _rtr := _rtrStateless;
            _stop := _stopStateless;
            conv := convStateless;
            eq := eqStateless;
            stopsensor := stopsensorStateless;
            nextConv := nextConvStateless;
            prevConv := prevConvStateless;
        END_METHOD

        METHOD PUBLIC Setup
            _rtd.equipment := eq;
            _rtd.NextReceiver := nextConv;
            _rtd.StopPosition := _stop;
            _rtr.StopPosition := conv;
            _rtr.equipment := eq;
            _stop.StopSensor := stopsensor;
            _stop.Equipment := eq;
            _stop.Deliverer := _rtd;
            ;
        END_METHOD
        {Test}
        METHOD PUBLIC ReadyToDeliver_Is_True_when_conveyor_is_occupied_and_autostarted
            // Arrange - Setup transport control logic with occupied conveyor
            THIS.Setup();
            nextConv.RTR := ReceiveState#ReadyToReceive;  // Next conveyor ready
            eq.MockStatus := StartUpStatus#AutoStartedUp;  // Equipment auto-started
            stopsensor.QValue := TRUE;  // Stop sensor covered (item present)

            // Act - First evaluation cycle
            _stop.EvaluateStopPos();
            _internalDeliverState := _rtd.EvaluateDeliverStatus();
            _internalReceiveState := _rtr.EvaluateReceiveStatus();

            // Assert - Transfer should be in progress, ready to receive
            Equal(expected := TRUE, actual := _internalDeliverState = DeliverState#Delivering);
            Equal(expected := TRUE, actual := _internalReceiveState = ReceiveState#ReadyToReceive);

            // Act - Second evaluation cycle (verify state persistence)
            _stop.EvaluateStopPos();
            _internalDeliverState := _rtd.EvaluateDeliverStatus();
            _internalReceiveState := _rtr.EvaluateReceiveStatus();

            // Assert - States should remain consistent
            Equal(expected := TRUE, actual := _internalDeliverState = DeliverState#Delivering);
            Equal(expected := TRUE, actual := _internalReceiveState = ReceiveState#ReadyToReceive);

            // Act - Third evaluation cycle (verify continued stability)
            _stop.EvaluateStopPos();
            _internalDeliverState := _rtd.EvaluateDeliverStatus();
            _internalReceiveState := _rtr.EvaluateReceiveStatus();

            // Assert - States should still be consistent across multiple cycles
            Equal(expected := TRUE, actual := _internalDeliverState = DeliverState#Delivering);
            Equal(expected := TRUE, actual := _internalReceiveState = ReceiveState#ReadyToReceive);

        END_METHOD

    END_CLASS

END_NAMESPACE

(* ---- TransportToNextConveyorTest.st ---- *)
USING Simatic.Ax.Conveyor.Mocks;
USING Simatic.Ax.Conveyor;
USING AxUnit.Assert;
USING Simatic.Ax.AutomationBase;
USING MotorTests.Mocks;

NAMESPACE Simatic.Ax.Conveyor

    /// Tests for transporting items to next conveyor
    /// Verifies coordination between conveyors using ReadyToReceive signals
    {TestFixture}
    CLASS TransportToNextConveyorTest
        VAR
            conv : ConveyorBase;
            convStateless : ConveyorBase;
            nextConv : MockingConveyor;
            nextConvStateless : MockingConveyor;
            sensor : MockBinSignal;
            sensorStateless : MockBinSignal;
            relTrue : MockIsReleased_TRUE;
            relTrueStateless : MockIsReleased_TRUE;
            relFalse : MockIsReleased_FALSE;
            relFalseStateless : MockIsReleased_FALSE;
            autoStart : MockAutoStartup := (startupStatus := StartUpStatus#AutoStartedUp);
            autoStartStateless : MockAutoStartup := (startupStatus := StartUpStatus#AutoStartedUp);
            mode : MockOperatingMode;
            modeStateless : MockOperatingMode;
            mockMotor : MockMotor;
            mockMotorStateless : MockMotor;
        END_VAR

        {TestSetup}
        METHOD PUBLIC TestSetup
            // Initialize stateless instances for each test
            conv := convStateless;
            nextConv := nextConvStateless;
            sensor := sensorStateless;
            relTrue := relTrueStateless;
            relFalse := relFalseStateless;
            autoStart := autoStartStateless;
            mode := modeStateless;
            mockMotor := mockMotorStateless;
            mockMotor.Reset();

            // Setup conveyor configuration
            conv.NextConveyor := nextConv;
            conv.StopSensor := sensor;
            conv.Motor := mockMotor;
            conv.ExternalRelease := relTrue;
            conv.ExternalAutoStartup := autoStart;
            conv.Mode := mode;
            mode.mode := OperatingModes#Automatic;
            AxUnit.Mocking.Mock('System.Timer.OffDelay', 'Simatic.Ax.Mocks.OffDelayMock_pass_trough');
        END_METHOD

        {Test}
        METHOD PUBLIC Fully_released_Conveyor_is_running_when_Sensor_is_occupied_and_enxt_conv_is_ready_to_receive
            // Arrange - Setup conveyor with sensor covered and next conveyor ready
            nextConv.RTR := ReceiveState#ReadyToReceive;
            sensor.QValue := TRUE;  // Item on sensor

            // Act - Run cyclic execution
            conv.RunCyclic();

            // Assert - Motor should be running and transfer in progress
            Equal(expected := TRUE, actual := mockMotor.IsRunning());
            Equal(expected := TRUE, actual := conv.DeliverStatus() = DeliverState#Delivering);

            // Act - Continue running multiple cycles
            conv.RunCyclic();

            // Assert - Motor should remain running
            Equal(expected := TRUE, actual := mockMotor.IsRunning());

            conv.RunCyclic();
            Equal(expected := TRUE, actual := mockMotor.IsRunning());

            conv.RunCyclic();
            Equal(expected := TRUE, actual := mockMotor.IsRunning());
        END_METHOD

        {Test}
        METHOD PUBLIC Fully_released_and_running_Conveyor_stops_when_Sensor_is_occupied_and_next_conveyor_looses_RTR
            // Arrange - Setup conveyor running with transfer in progress
            THIS.Fully_released_Conveyor_is_running_when_Sensor_is_occupied_and_enxt_conv_is_ready_to_receive();

            // Verify motor is running
            Equal(expected := TRUE, actual := mockMotor.IsRunning());

            // Act - Next conveyor loses ready to receive signal
            nextConv.RTR := ReceiveState#Idle;
            sensor.QValue := TRUE;  // Item still on sensor
            conv.RunCyclic();

            // Assert - Motor should stop when next conveyor is not ready
            Equal(expected := FALSE, actual := mockMotor.IsRunning());
        END_METHOD

        {Test}
        METHOD PUBLIC Stopped_and_empty_Conveyor_Starts_After_first_sensor_is_covered_and_then_rtr_becomes_true
            // Arrange - Setup stopped conveyor with next conveyor not ready
            nextConv.RTR := ReceiveState#Idle;
            sensor.QValue := FALSE;

            // Run once to complete startup and move to basic position
            conv.RunCyclic();

            // Act - Simulate home position run completed (off delay expires)
            AxUnit.Mocking.Mock('System.Timer.OffDelay', 'Simatic.Ax.Mocks.OffDelayMock_false');
            conv.RunCyclic();

            // Assert - Motor should be stopped after home position
            Equal(expected := FALSE, actual := mockMotor.IsRunning());

            // Act - Item arrives on sensor (but next conveyor not ready yet)
            sensor.QValue := TRUE;
            conv.RunCyclic();

            // Assert - Motor should remain stopped, but conveyor is occupied
            Equal(expected := FALSE, actual := mockMotor.IsRunning());
            Equal(expected := TRUE, actual := conv.IsOccupied());

            // Act - Next conveyor becomes ready to receive
            nextConv.RTR := ReceiveState#ReadyToReceive;
            AxUnit.Mocking.Mock('System.Timer.OffDelay', 'Simatic.Ax.Mocks.OffDelayMock_true');
            conv.RunCyclic();

            // Assert - Motor should start now that both conditions are met
            Equal(expected := TRUE, actual := mockMotor.IsRunning());
        END_METHOD

        {Test}
        METHOD PUBLIC Stopped_and_empty_Conveyor_Starts_After_rtr_true_and_then_sensor_becomes_covered
            // Arrange - Setup stopped conveyor with next conveyor not ready
            nextConv.RTR := ReceiveState#Idle;
            sensor.QValue := FALSE;

            // Run once to complete startup and move to basic position
            conv.RunCyclic();

            // Act - Simulate home position run completed (off delay expires)
            AxUnit.Mocking.Mock('System.Timer.OffDelay', 'Simatic.Ax.Mocks.OffDelayMock_false');
            conv.RunCyclic();

            // Assert - Motor should be stopped after home position
            Equal(expected := FALSE, actual := mockMotor.IsRunning());

            // Act - Next conveyor becomes ready (but no item yet)
            nextConv.RTR := ReceiveState#ReadyToReceive;
            conv.RunCyclic();

            // Assert - Motor should remain stopped without item
            Equal(expected := FALSE, actual := mockMotor.IsRunning());

            // Act - Item arrives on sensor
            sensor.QValue := TRUE;
            AxUnit.Mocking.Mock('System.Timer.OffDelay', 'System.Timer.OffDelay');
            conv.RunCyclic();

            // Assert - Conveyor should be occupied and transfer in progress
            Equal(expected := TRUE, actual := conv.IsOccupied());
            Equal(expected := TRUE, actual := conv.Delivering());
            Equal(expected := TRUE, actual := mockMotor.IsRunning());

            // Act - Item leaves sensor (transfer complete)
            sensor.QValue := FALSE;
            conv.RunCyclic();

            // Assert - Transfer finished, conveyor no longer occupied
            Equal(expected := FALSE, actual := conv.Delivering());
            Equal(expected := FALSE, actual := conv.IsOccupied());
        END_METHOD

        {Test}
        METHOD PUBLIC Conveyor_is_stopped__when_in_inAutomatic_but_without_release
            // Arrange - Setup conveyor in automatic mode without release
            conv.ExternalRelease := relFalse;  // No release signal
            autoStart.startupStatus := StartUpStatus#NotReleased;

            // Verify configuration is valid
            Equal(expected := FALSE, actual := HasConfigErrorTest(eq := conv));

            // Act - Run cyclic execution
            conv.RunCyclic();

            // Assert - Motor should not run without release signal
            Equal(expected := FALSE, actual := mockMotor.IsRunning());
        END_METHOD
    END_CLASS

END_NAMESPACE
